// SIMATIC S7-200 SMART project (STEP 7-Micro/WIN SMART), CPU ST60

SYMBOL_TABLE 系统符号
Always_On        SM0.0    // 始终接通
END_SYMBOL_TABLE

ORGANIZATION_BLOCK MAIN:OB1
TITLE=程序注释
BEGIN
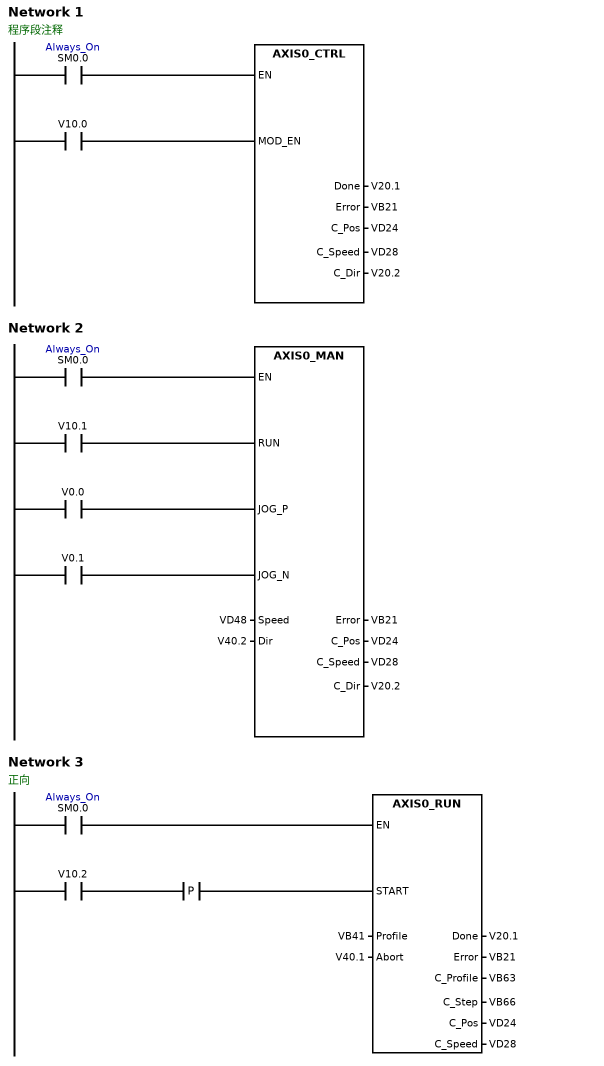
Network 1
// 程序段注释
LD     Always_On:SM0.0
=      L60.0
LD     V10.0
=      L63.7
LD     L60.0
CALL   AXIS0_CTRL:SBR1, L63.7, V20.1, VB21, VD24, VD28, V20.2
Network 2
LD     Always_On:SM0.0
=      L60.0
LD     V10.1
=      L63.7
LD     V0.0
=      L63.6
LD     V0.1
=      L63.5
LD     L60.0
CALL   AXIS0_MAN:SBR2, L63.7, L63.6, L63.5, VD48, V40.2, VB21, VD24, VD28, V20.2
Network 3
// 正向
LD     Always_On:SM0.0
=      L60.0
LD     V10.2
EU
=      L63.7
LD     L60.0
CALL   AXIS0_RUN:SBR4, L63.7, VB41, V40.1, V20.1, VB21, VB63, VB66, VD24, VD28
END_ORGANIZATION_BLOCK

// SBR1: protected block, not included

// SBR2: protected block, not included

// SBR3: protected block, not included

// SBR4: protected block, not included

// SBR5: protected block, not included

// SBR6: protected block, not included

// SBR7: protected block, not included

// SBR8: protected block, not included

// SBR9: protected block, not included

// SBR10: protected block, not included

// SBR11: protected block, not included
